TYPE ParallelUnitsSettings :
STRUCT
	RemoteAmsId: STRING := '5.73.47.143.1.1';
	PressureSupplySP: LREAL := 250; // Set Point for Master/Slave
	PressureExtractSP: LREAL := 280; // Set Point for Master/Slave
	PressureSupplySP_HighSpeed: LREAL := 275; // Set Point for Master/Slave
	PressureExtractSP_HighSpeed: LREAL := 295; // Set Point for Master/Slave
	StandaloneMaxFan: LREAL := 0.7; // Max fan speed for single unit
	DualMinFan: LREAL := 0.4; // Min fan speed for dual units
	Kp: LREAL := 1.5; // P
	fTn: TIME := T#4M; // I time
	fTv: TIME := T#0M; // D time
	RemoteOrder: RemoteOrder;
	StandalonePressureSupplySP: LREAL := 125;
	StandalonePressureExtractSP: LREAL := 150;
	StandalonePressureSupplySP_HighSpeed: LREAL := 150;
	StandalonePressureExtractSP_HighSpeed: LREAL := 175;
END_STRUCT
END_TYPE

(* stored: Version 1.1.0.1, ProductVersion 3.1.4024.6
   DUT ParallelUnitsSettings: Id {be21b28a-d10a-4ec1-8077-12ca649c2986} *)
